// TIA Portal project "项目12" (V18)

(* hardware
DEVICE "S7-1500/ET200MP station_1"  S7-1500 station
   slot 0: "导轨_0"  Rack  6ES7 590-1***0-0AA0
   slot 1: "PLC_1"  Unspecific CPU 1500  6ES7 5XX-XXXXX-XXXX  V3.0
*)

// ===== PLC "PLC_1"  Unspecific CPU 1500 =====

VAR_GLOBAL   // PLC tag table "默认变量表"
   "GDSR" AT %I0.2 : Bool;   // 光电传感器(右)
   "GDSL" AT %I0.3 : Bool;   // 光电传感器(左)
   "B_AN" AT %I1.0 : Bool;   // 蓝色按钮
   "G_AN" AT %I1.1 : Bool;   // 绿色按钮
   "Y_AN" AT %I1.2 : Bool;   // 黄色按钮
   "R_AN" AT %I1.3 : Bool;   // 红色按钮
   "ST_AN" AT %I1.4 : Bool;   // 急停按钮
   "PDZZ" AT %Q0.0 : Bool;   // 皮带正转
   "PDFZ" AT %Q0.1 : Bool;   // 皮带反转
   "B_L" AT %Q1.0 : Bool;   // 蓝灯
   "G_L" AT %Q1.1 : Bool;   // 绿灯
   "Y_L" AT %Q1.2 : Bool;   // 黄灯
   "R_L" AT %Q1.3 : Bool;   // 红灯
   "启动条件" AT %M10.0 : Bool;   // 启动条件
END_VAR

ORGANIZATION_BLOCK "Main"   // OB1, LAD, ProgramCycle
TITLE = "Main Program Sweep (Cycle)"
{ S7_Optimized_Access := 'TRUE' }
VERSION : 0.1
   VAR_INPUT
      Initial_Call : Bool;   // Initial call of this OB
      Remanence : Bool;   // =True, if remanent data are available
   END_VAR
BEGIN

REGION Network 1: 启动条件
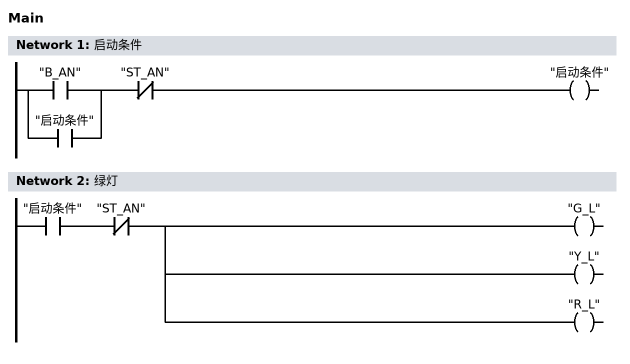
   RUNG wire#powerrail
      Contact( "B_AN" )
      wire#w1
      I_Contact( "ST_AN" )
      Coil( "启动条件" )
   END_RUNG
   RUNG wire#powerrail
      Contact( "启动条件" )
   END_RUNG wire#w1
   // the same network as SCL:
   "启动条件" := ("B_AN" OR "启动条件") AND NOT "ST_AN";
END_REGION

REGION Network 2: 绿灯
   RUNG wire#powerrail
      Contact( "启动条件" )
      I_Contact( "ST_AN" )
      wire#w1
      Coil( "G_L" )
   END_RUNG
   RUNG wire#w1
      Coil( "Y_L" )
   END_RUNG
   RUNG wire#w1
      Coil( "R_L" )
   END_RUNG
   // the same network as SCL:
   "G_L" := "启动条件" AND NOT "ST_AN";
   "Y_L" := "G_L";
   "R_L" := "G_L";
END_REGION
END_ORGANIZATION_BLOCK